Fanuc KAREL source: ka00133.KL

-- PROVISIONAL review KL for V1013-1; original PC SHA256 67aaee2939b66e57343fee75fb6e9c6ecaff3b5f60c147f511203e600b870c9a
-- Incomplete behavior may be omitted. Consult companion uncertainty JSON. Do not deploy.
PROGRAM KA00133
%NOLOCKGROUP
VAR
  DST : INTEGER
-- UNRESOLVED_DECL SRC type=002017
BEGIN
  -- UNRESOLVED_PC offsets 5-19; opcodes 2E,22,9D,33,B4
  -- UNRESOLVED_PC offsets 24-39; opcodes 22,9D,33,B3,23
  -- UNRESOLVED_PC offsets 44-48; opcodes 7F
END KA00133
